FUNCTION_BLOCK FB_Variante IMPLEMENTS I_Derived
VAR_INPUT
END_VAR
VAR_OUTPUT
END_VAR
VAR
END_VAR

{warning 'add method implementation '}
METHOD Base : BOOL
END_METHOD

{warning 'add method implementation '}
METHOD Derived : BOOL
END_METHOD

END_FUNCTION_BLOCK

(* stored: Version 1.1.0.1, ProductVersion 3.1.4024.12
   POU FB_Variante: Id {b96cac43-7242-4a32-9ec2-8d0f27d09c40}, SpecialFunc None
   Method Base: Id {8bc0bc5b-dac6-450a-88a6-2701749687ee}
   Method Derived: Id {bb0be15b-958a-4a61-9e22-3bbb210b7faf} *)
